FUNCTION alg_g_z: LREAL
VAR_INPUT
    state: STATE;
END_VAR

alg_g_z := state.curTime;

END_FUNCTION

(* stored: ProductVersion 3.1.0.18, Version 1.1.0.1 *)
